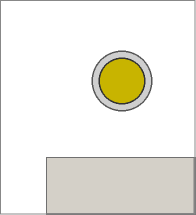
VISUALIZATION Visualization  // 196x215
    Button (46,157 150x58)
        tap MAIN.xInput
    Lamp1 (87,46 70x70), variable: MAIN.xOutput, style: Lamp-Lamp1-Yellow
END_VISUALIZATION

(* stored: Version 1.1.0.1, ProductVersion 3.1.4024.12
   Visu Visualization: Id {003a4796-faca-4859-b29a-b2047c367123} *)
